PROGRAM MAIN
VAR
    {attribute 'pytmc' := '
      pv: VCN:TEST:01
     '}
	fbVCN590 : FB_VCN_VAT590; // Variable leak valve function block
END_VAR

fbVCN590(i_xExtIlkOK := TRUE);

END_PROGRAM

(* stored: Version 1.1.0.1, ProductVersion 3.1.4024.6
   POU MAIN: Id {e705ade6-0f0a-4b24-98f0-3b81c602a7eb}, SpecialFunc None *)
